// TIA Portal V18 export
DATA_BLOCK "HWModulesConf"   // DB10002
{ S7_Optimized_Access := 'TRUE' }
VERSION : 0.1
// stored: AutoNumber false, DBAccessibleFromOPCUA true, IsOnlyStoredInLoadMemory false, IsRetainMemResEnabled false, IsWriteProtectedInAS false, MemoryReserve 100
   VAR
      HW { S7_SetPoint := 'True'} : Array[1..14] of "UDT_HWModulesMap";
   END_VAR
BEGIN
   HW[1..8].cRack := 11;
   HW[9..14].cRack := 12;
   HW[1].cModule := 1;
   HW[2].cModule := 2;
   HW[3].cModule := 3;
   HW[4].cModule := 4;
   HW[5].cModule := 5;
   HW[6].cModule := 6;
   HW[7..8].cModule := 7;
   HW[9].cModule := 0;
   HW[10].cModule := 1;
   HW[11].cModule := 2;
   HW[12].cModule := 3;
   HW[13].cModule := 4;
   HW[14].cModule := 5;
   HW[1].wLaddr1 := 263;
   HW[2].wLaddr1 := 269;
   HW[3].wLaddr1 := 270;
   HW[4].wLaddr1 := 286;
   HW[5].wLaddr1 := 271;
   HW[6].wLaddr1 := 272;
   HW[7].wLaddr1 := 287;
   HW[8].wLaddr1 := 288;
   HW[9].wLaddr1 := 280;
   HW[10].wLaddr1 := 282;
   HW[11].wLaddr1 := 283;
   HW[12].wLaddr1 := 284;
   HW[13].wLaddr1 := 285;
   HW[14].wLaddr1 := 281;
   HW[1].wLaddr2 := 264;
END_DATA_BLOCK
